// TIA Portal V19 export
FUNCTION "FC60_Fault" : Void   // FC60, LAD
{ S7_Optimized_Access := 'TRUE' }
// stored: AutoNumber false, IsIECCheckEnabled true, SetENOAutomatically false
   VAR_TEMP
      txFaultMaster : Bool;
      txFaultLeft : Bool;
      txFaultRight : Bool;
   END_VAR
BEGIN

REGION Network 1: Safety fault
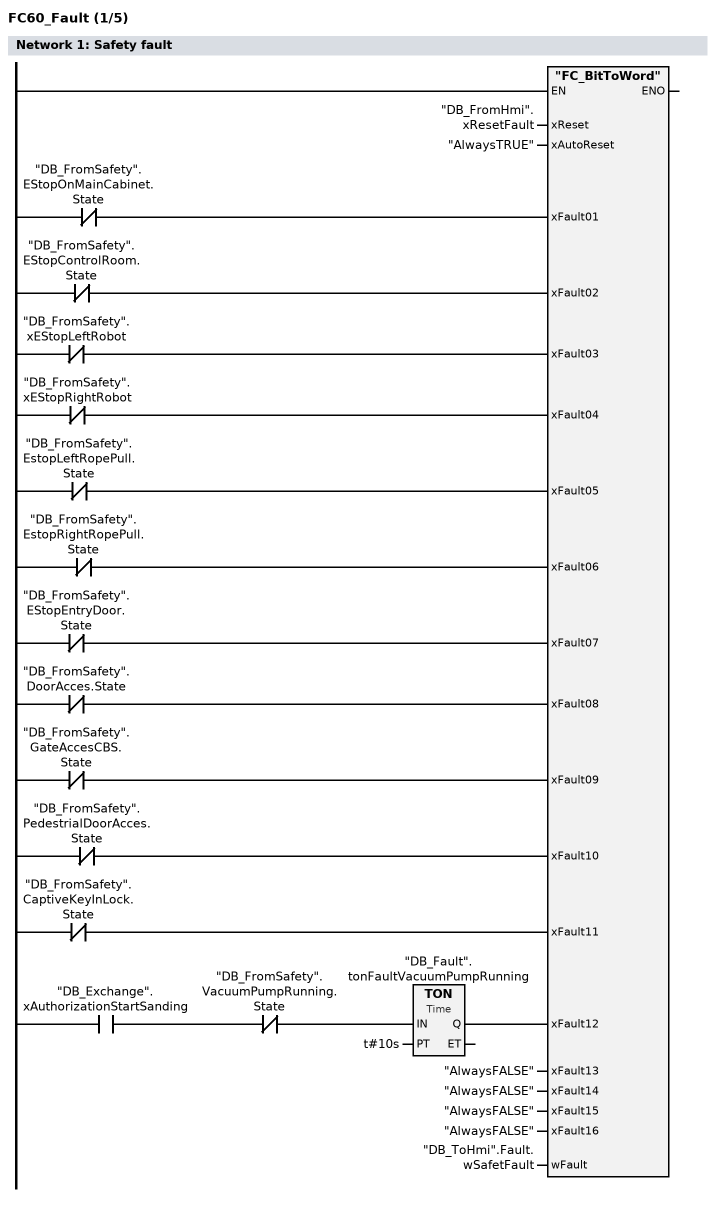
   RUNG wire#powerrail
      "FC_BitToWord"(xFault01 := wire#w1, xFault02 := wire#w2, xFault03 := wire#w3, xFault04 := wire#w4, xFault05 := wire#w5, xFault06 := wire#w6, xFault07 := wire#w7, xFault08 := wire#w8, xFault09 := wire#w9, xFault10 := wire#w10, xFault11 := wire#w11, xFault12 := wire#w12, xReset := "DB_FromHmi".xResetFault, xAutoReset := "AlwaysTRUE", xFault13 := "AlwaysFALSE", xFault14 := "AlwaysFALSE", xFault15 := "AlwaysFALSE", xFault16 := "AlwaysFALSE", wFault := "DB_ToHmi".Fault.wSafetFault)
   END_RUNG
   RUNG wire#powerrail
      I_Contact( "DB_FromSafety".EStopOnMainCabinet.State )
   END_RUNG wire#w1
   RUNG wire#powerrail
      I_Contact( "DB_FromSafety".EStopControlRoom.State )
   END_RUNG wire#w2
   RUNG wire#powerrail
      I_Contact( "DB_FromSafety".xEStopLeftRobot )
   END_RUNG wire#w3
   RUNG wire#powerrail
      I_Contact( "DB_FromSafety".xEStopRightRobot )
   END_RUNG wire#w4
   RUNG wire#powerrail
      I_Contact( "DB_FromSafety".EstopLeftRopePull.State )
   END_RUNG wire#w5
   RUNG wire#powerrail
      I_Contact( "DB_FromSafety".EstopRightRopePull.State )
   END_RUNG wire#w6
   RUNG wire#powerrail
      I_Contact( "DB_FromSafety".EStopEntryDoor.State )
   END_RUNG wire#w7
   RUNG wire#powerrail
      I_Contact( "DB_FromSafety".DoorAcces.State )
   END_RUNG wire#w8
   RUNG wire#powerrail
      I_Contact( "DB_FromSafety".GateAccesCBS.State )
   END_RUNG wire#w9
   RUNG wire#powerrail
      I_Contact( "DB_FromSafety".PedestrialDoorAcces.State )
   END_RUNG wire#w10
   RUNG wire#powerrail
      I_Contact( "DB_FromSafety".CaptiveKeyInLock.State )
   END_RUNG wire#w11
   RUNG wire#powerrail
      Contact( "DB_Exchange".xAuthorizationStartSanding )
      I_Contact( "DB_FromSafety".VacuumPumpRunning.State )
      { S7_Templates := "time_type := Time" } "DB_Fault".tonFaultVacuumPumpRunning.TON(pt := t#10s, et =>)
   END_RUNG wire#w12
   // the same network as SCL:
   "DB_Fault".tonFaultVacuumPumpRunning.TON(IN := "DB_Exchange".xAuthorizationStartSanding AND NOT "DB_FromSafety".VacuumPumpRunning.State,
                           PT := t#10s);
   "FC_BitToWord"(xReset := "DB_FromHmi".xResetFault,
                  xAutoReset := "AlwaysTRUE",
                  xFault01 := NOT "DB_FromSafety".EStopOnMainCabinet.State,
                  xFault02 := NOT "DB_FromSafety".EStopControlRoom.State,
                  xFault03 := NOT "DB_FromSafety".xEStopLeftRobot,
                  xFault04 := NOT "DB_FromSafety".xEStopRightRobot,
                  xFault05 := NOT "DB_FromSafety".EstopLeftRopePull.State,
                  xFault06 := NOT "DB_FromSafety".EstopRightRopePull.State,
                  xFault07 := NOT "DB_FromSafety".EStopEntryDoor.State,
                  xFault08 := NOT "DB_FromSafety".DoorAcces.State,
                  xFault09 := NOT "DB_FromSafety".GateAccesCBS.State,
                  xFault10 := NOT "DB_FromSafety".PedestrialDoorAcces.State,
                  xFault11 := NOT "DB_FromSafety".CaptiveKeyInLock.State,
                  xFault12 := "DB_Fault".tonFaultVacuumPumpRunning.Q,
                  xFault13 := "AlwaysFALSE",
                  xFault14 := "AlwaysFALSE",
                  xFault15 := "AlwaysFALSE",
                  xFault16 := "AlwaysFALSE",
                  wFault := "DB_ToHmi".Fault.wSafetFault);
END_REGION

REGION Network 2: Error safety module
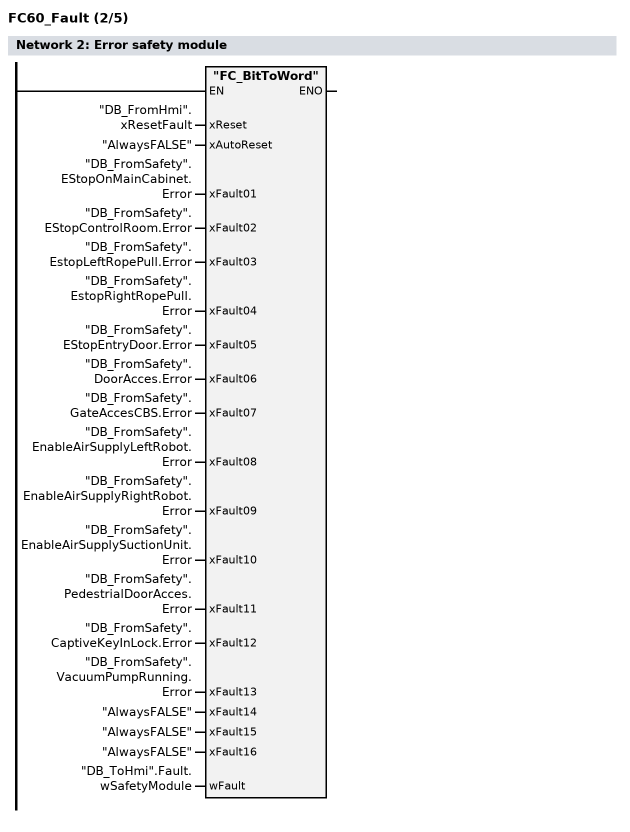
   RUNG wire#powerrail
      "FC_BitToWord"(xReset := "DB_FromHmi".xResetFault, xAutoReset := "AlwaysFALSE", xFault01 := "DB_FromSafety".EStopOnMainCabinet.Error, xFault02 := "DB_FromSafety".EStopControlRoom.Error, xFault03 := "DB_FromSafety".EstopLeftRopePull.Error, xFault04 := "DB_FromSafety".EstopRightRopePull.Error, xFault05 := "DB_FromSafety".EStopEntryDoor.Error, xFault06 := "DB_FromSafety".DoorAcces.Error, xFault07 := "DB_FromSafety".GateAccesCBS.Error, xFault08 := "DB_FromSafety".EnableAirSupplyLeftRobot.Error, xFault09 := "DB_FromSafety".EnableAirSupplyRightRobot.Error, xFault10 := "DB_FromSafety".EnableAirSupplySuctionUnit.Error, xFault11 := "DB_FromSafety".PedestrialDoorAcces.Error, xFault12 := "DB_FromSafety".CaptiveKeyInLock.Error, xFault13 := "DB_FromSafety".VacuumPumpRunning.Error, xFault14 := "AlwaysFALSE", xFault15 := "AlwaysFALSE", xFault16 := "AlwaysFALSE", wFault := "DB_ToHmi".Fault.wSafetyModule)
   END_RUNG
   // the same network as SCL:
   "FC_BitToWord"(xReset := "DB_FromHmi".xResetFault,
                  xAutoReset := "AlwaysFALSE",
                  xFault01 := "DB_FromSafety".EStopOnMainCabinet.Error,
                  xFault02 := "DB_FromSafety".EStopControlRoom.Error,
                  xFault03 := "DB_FromSafety".EstopLeftRopePull.Error,
                  xFault04 := "DB_FromSafety".EstopRightRopePull.Error,
                  xFault05 := "DB_FromSafety".EStopEntryDoor.Error,
                  xFault06 := "DB_FromSafety".DoorAcces.Error,
                  xFault07 := "DB_FromSafety".GateAccesCBS.Error,
                  xFault08 := "DB_FromSafety".EnableAirSupplyLeftRobot.Error,
                  xFault09 := "DB_FromSafety".EnableAirSupplyRightRobot.Error,
                  xFault10 := "DB_FromSafety".EnableAirSupplySuctionUnit.Error,
                  xFault11 := "DB_FromSafety".PedestrialDoorAcces.Error,
                  xFault12 := "DB_FromSafety".CaptiveKeyInLock.Error,
                  xFault13 := "DB_FromSafety".VacuumPumpRunning.Error,
                  xFault14 := "AlwaysFALSE",
                  xFault15 := "AlwaysFALSE",
                  xFault16 := "AlwaysFALSE",
                  wFault := "DB_ToHmi".Fault.wSafetyModule);
END_REGION

REGION Network 3: Other fault on Master PLC
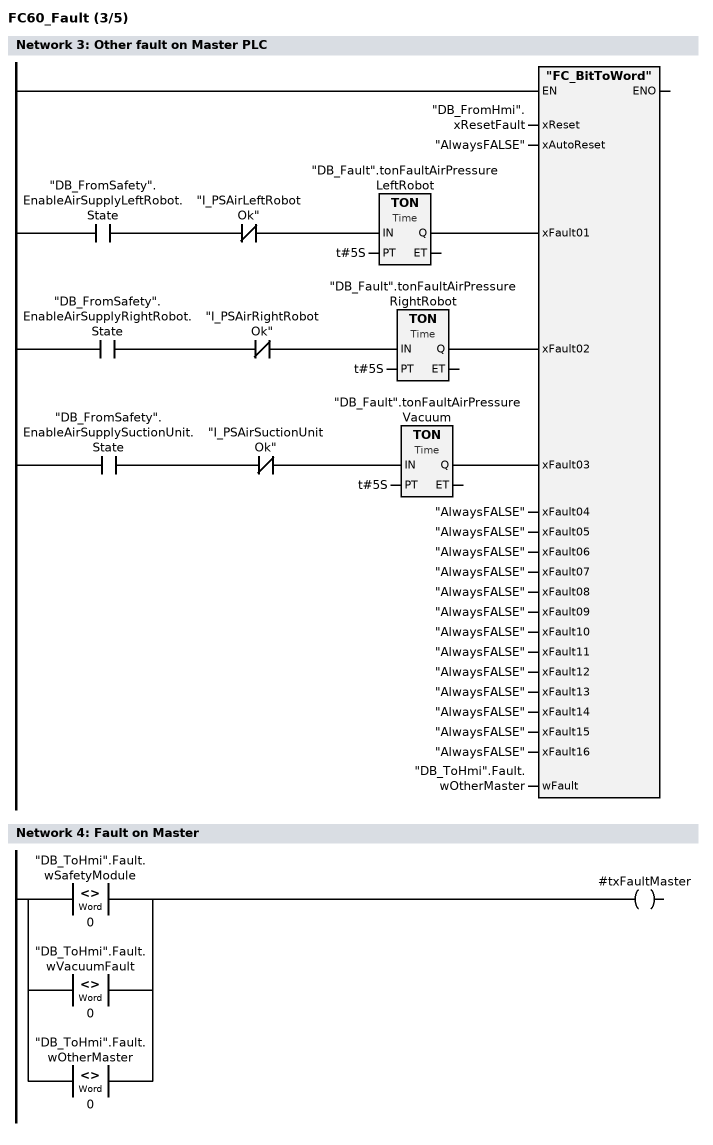
   RUNG wire#powerrail
      "FC_BitToWord"(xFault01 := wire#w1, xFault02 := wire#w2, xFault03 := wire#w3, xReset := "DB_FromHmi".xResetFault, xAutoReset := "AlwaysFALSE", xFault04 := "AlwaysFALSE", xFault05 := "AlwaysFALSE", xFault06 := "AlwaysFALSE", xFault07 := "AlwaysFALSE", xFault08 := "AlwaysFALSE", xFault09 := "AlwaysFALSE", xFault10 := "AlwaysFALSE", xFault11 := "AlwaysFALSE", xFault12 := "AlwaysFALSE", xFault13 := "AlwaysFALSE", xFault14 := "AlwaysFALSE", xFault15 := "AlwaysFALSE", xFault16 := "AlwaysFALSE", wFault := "DB_ToHmi".Fault.wOtherMaster)
   END_RUNG
   RUNG wire#powerrail
      Contact( "DB_FromSafety".EnableAirSupplyLeftRobot.State )
      I_Contact( "I_PSAirLeftRobotOk" )
      { S7_Templates := "time_type := Time" } "DB_Fault".tonFaultAirPressureLeftRobot.TON(pt := t#5S, et =>)
   END_RUNG wire#w1
   RUNG wire#powerrail
      Contact( "DB_FromSafety".EnableAirSupplyRightRobot.State )
      I_Contact( "I_PSAirRightRobotOk" )
      { S7_Templates := "time_type := Time" } "DB_Fault".tonFaultAirPressureRightRobot.TON(pt := t#5S, et =>)
   END_RUNG wire#w2
   RUNG wire#powerrail
      Contact( "DB_FromSafety".EnableAirSupplySuctionUnit.State )
      I_Contact( "I_PSAirSuctionUnitOk" )
      { S7_Templates := "time_type := Time" } "DB_Fault".tonFaultAirPressureVacuum.TON(pt := t#5S, et =>)
   END_RUNG wire#w3
   // the same network as SCL:
   "DB_Fault".tonFaultAirPressureLeftRobot.TON(IN := "DB_FromSafety".EnableAirSupplyLeftRobot.State AND NOT "I_PSAirLeftRobotOk",
                           PT := t#5S);
   "DB_Fault".tonFaultAirPressureRightRobot.TON(IN := "DB_FromSafety".EnableAirSupplyRightRobot.State AND NOT "I_PSAirRightRobotOk",
                           PT := t#5S);
   "DB_Fault".tonFaultAirPressureVacuum.TON(IN := "DB_FromSafety".EnableAirSupplySuctionUnit.State AND NOT "I_PSAirSuctionUnitOk",
                           PT := t#5S);
   "FC_BitToWord"(xReset := "DB_FromHmi".xResetFault,
                  xAutoReset := "AlwaysFALSE",
                  xFault01 := "DB_Fault".tonFaultAirPressureLeftRobot.Q,
                  xFault02 := "DB_Fault".tonFaultAirPressureRightRobot.Q,
                  xFault03 := "DB_Fault".tonFaultAirPressureVacuum.Q,
                  xFault04 := "AlwaysFALSE",
                  xFault05 := "AlwaysFALSE",
                  xFault06 := "AlwaysFALSE",
                  xFault07 := "AlwaysFALSE",
                  xFault08 := "AlwaysFALSE",
                  xFault09 := "AlwaysFALSE",
                  xFault10 := "AlwaysFALSE",
                  xFault11 := "AlwaysFALSE",
                  xFault12 := "AlwaysFALSE",
                  xFault13 := "AlwaysFALSE",
                  xFault14 := "AlwaysFALSE",
                  xFault15 := "AlwaysFALSE",
                  xFault16 := "AlwaysFALSE",
                  wFault := "DB_ToHmi".Fault.wOtherMaster);
END_REGION

REGION Network 4: Fault on Master
   RUNG wire#powerrail
      { S7_Templates := "SrcType := Word" } NE_Contact(in1 := "DB_ToHmi".Fault.wSafetyModule, in2 := 0)
      wire#w1
      Coil( #txFaultMaster )
   END_RUNG
   RUNG wire#powerrail
      { S7_Templates := "SrcType := Word" } NE_Contact(in1 := "DB_ToHmi".Fault.wVacuumFault, in2 := 0)
   END_RUNG wire#w1
   RUNG wire#powerrail
      { S7_Templates := "SrcType := Word" } NE_Contact(in1 := "DB_ToHmi".Fault.wOtherMaster, in2 := 0)
   END_RUNG wire#w1
   // the same network as SCL:
   #txFaultMaster := ("DB_ToHmi".Fault.wSafetyModule <> 0) OR ("DB_ToHmi".Fault.wVacuumFault <> 0) OR ("DB_ToHmi".Fault.wOtherMaster <> 0);
END_REGION

REGION Network 5: Fault on Left
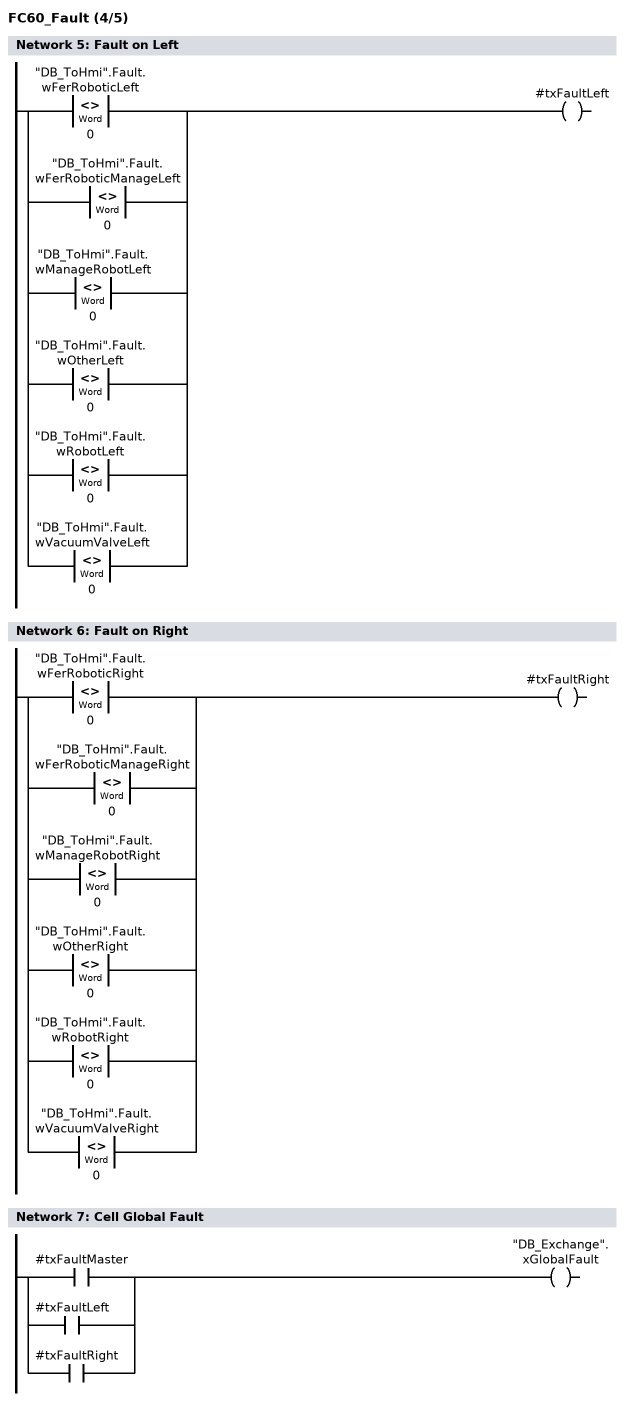
   RUNG wire#powerrail
      { S7_Templates := "SrcType := Word" } NE_Contact(in1 := "DB_ToHmi".Fault.wFerRoboticLeft, in2 := 0)
      wire#w1
      Coil( #txFaultLeft )
   END_RUNG
   RUNG wire#powerrail
      { S7_Templates := "SrcType := Word" } NE_Contact(in1 := "DB_ToHmi".Fault.wFerRoboticManageLeft, in2 := 0)
   END_RUNG wire#w1
   RUNG wire#powerrail
      { S7_Templates := "SrcType := Word" } NE_Contact(in1 := "DB_ToHmi".Fault.wManageRobotLeft, in2 := 0)
   END_RUNG wire#w1
   RUNG wire#powerrail
      { S7_Templates := "SrcType := Word" } NE_Contact(in1 := "DB_ToHmi".Fault.wOtherLeft, in2 := 0)
   END_RUNG wire#w1
   RUNG wire#powerrail
      { S7_Templates := "SrcType := Word" } NE_Contact(in1 := "DB_ToHmi".Fault.wRobotLeft, in2 := 0)
   END_RUNG wire#w1
   RUNG wire#powerrail
      { S7_Templates := "SrcType := Word" } NE_Contact(in1 := "DB_ToHmi".Fault.wVacuumValveLeft, in2 := 0)
   END_RUNG wire#w1
   // the same network as SCL:
   #txFaultLeft := ("DB_ToHmi".Fault.wFerRoboticLeft <> 0) OR ("DB_ToHmi".Fault.wFerRoboticManageLeft <> 0) OR ("DB_ToHmi".Fault.wManageRobotLeft <> 0) OR ("DB_ToHmi".Fault.wOtherLeft <> 0) OR ("DB_ToHmi".Fault.wRobotLeft <> 0) OR ("DB_ToHmi".Fault.wVacuumValveLeft <> 0);
END_REGION

REGION Network 6: Fault on Right
   RUNG wire#powerrail
      { S7_Templates := "SrcType := Word" } NE_Contact(in1 := "DB_ToHmi".Fault.wFerRoboticRight, in2 := 0)
      wire#w1
      Coil( #txFaultRight )
   END_RUNG
   RUNG wire#powerrail
      { S7_Templates := "SrcType := Word" } NE_Contact(in1 := "DB_ToHmi".Fault.wFerRoboticManageRight, in2 := 0)
   END_RUNG wire#w1
   RUNG wire#powerrail
      { S7_Templates := "SrcType := Word" } NE_Contact(in1 := "DB_ToHmi".Fault.wManageRobotRight, in2 := 0)
   END_RUNG wire#w1
   RUNG wire#powerrail
      { S7_Templates := "SrcType := Word" } NE_Contact(in1 := "DB_ToHmi".Fault.wOtherRight, in2 := 0)
   END_RUNG wire#w1
   RUNG wire#powerrail
      { S7_Templates := "SrcType := Word" } NE_Contact(in1 := "DB_ToHmi".Fault.wRobotRight, in2 := 0)
   END_RUNG wire#w1
   RUNG wire#powerrail
      { S7_Templates := "SrcType := Word" } NE_Contact(in1 := "DB_ToHmi".Fault.wVacuumValveRight, in2 := 0)
   END_RUNG wire#w1
   // the same network as SCL:
   #txFaultRight := ("DB_ToHmi".Fault.wFerRoboticRight <> 0) OR ("DB_ToHmi".Fault.wFerRoboticManageRight <> 0) OR ("DB_ToHmi".Fault.wManageRobotRight <> 0) OR ("DB_ToHmi".Fault.wOtherRight <> 0) OR ("DB_ToHmi".Fault.wRobotRight <> 0) OR ("DB_ToHmi".Fault.wVacuumValveRight <> 0);
END_REGION

REGION Network 7: Cell Global Fault
   RUNG wire#powerrail
      Contact( #txFaultMaster )
      wire#w1
      Coil( "DB_Exchange".xGlobalFault )
   END_RUNG
   RUNG wire#powerrail
      Contact( #txFaultLeft )
   END_RUNG wire#w1
   RUNG wire#powerrail
      Contact( #txFaultRight )
   END_RUNG wire#w1
   // the same network as SCL:
   "DB_Exchange".xGlobalFault := #txFaultMaster OR #txFaultLeft OR #txFaultRight;
END_REGION

REGION Network 8: Cell Global warning
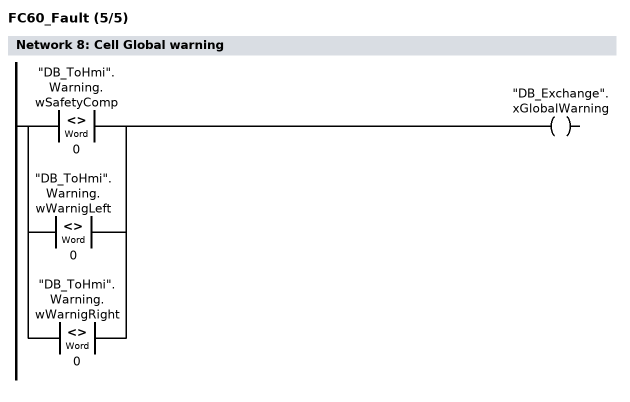
   RUNG wire#powerrail
      { S7_Templates := "SrcType := Word" } NE_Contact(in1 := "DB_ToHmi".Warning.wSafetyComp, in2 := 0)
      wire#w1
      Coil( "DB_Exchange".xGlobalWarning )
   END_RUNG
   RUNG wire#powerrail
      { S7_Templates := "SrcType := Word" } NE_Contact(in1 := "DB_ToHmi".Warning.wWarnigLeft, in2 := 0)
   END_RUNG wire#w1
   RUNG wire#powerrail
      { S7_Templates := "SrcType := Word" } NE_Contact(in1 := "DB_ToHmi".Warning.wWarnigRight, in2 := 0)
   END_RUNG wire#w1
   // the same network as SCL:
   "DB_Exchange".xGlobalWarning := ("DB_ToHmi".Warning.wSafetyComp <> 0) OR ("DB_ToHmi".Warning.wWarnigLeft <> 0) OR ("DB_ToHmi".Warning.wWarnigRight <> 0);
END_REGION
END_FUNCTION
